{attribute addProperty BoxType "EL3453-0000-0017"}
{attribute addProperty Id "FrequencyAT %I*REAL32417Power_FactorAT %I*REAL32418Calculated_Error_CurrentAT %I*REAL32420Neutral_Line_CurrentAT %I*REAL32421ROCOFAT %I*REAL32422"}
{attribute addProperty CRC "2480258228"}
{attribute addProperty SizeInBites "160"}
{attribute addProperty SizeInBytes "20"}
TYPE Total_Basic_93D5BCB4 :
STRUCT
	{attribute addProperty Name "Frequency"}
	Frequency AT %I* : REAL;
	{attribute addProperty Name "Power_Factor"}
	Power_Factor AT %I* : REAL;
	{attribute addProperty Name "Calculated_Error_Current"}
	Calculated_Error_Current AT %I* : REAL;
	{attribute addProperty Name "Neutral_Line_Current"}
	Neutral_Line_Current AT %I* : REAL;
	{attribute addProperty Name "ROCOF"}
	ROCOF AT %I* : REAL;
END_STRUCT
END_TYPE

(* stored: Version 1.2.0.0, ProductVersion 3.1.4024.9
   DUT Total_Basic_93D5BCB4: Id {82905ced-cb8a-4790-8859-70c644d7b277} *)
